(* CoDeSys 2.3.9.41 project: dct.pro *)
(* Libraries: STANDARD.LIB 4.10.05 11:14:46, IECSFC.LIB 13.4.06 15:51:28, SYSLIBTIME.LIB 20.2.06 13:31:16, SYSTASKINFO.LIB 20.2.06 13:31:38, ANALYZATION.LIB 5.10.99 09:05:06, SYSLIBCALLBACK.LIB 20.2.06 13:31:08 *)

(* PLC configuration (modules and I/O channels)
Discrete input 6 bit [ID100] node 0, in %IB0 out %QB0 {Filtrationtime = 10; Filtrationtime = 10; Filtrationtime = 10; Filtrationtime = 10; Filtrationtime = 10; Filtrationtime = 10; Visibility = No; PinCount = 6; WatchDogPeriod = 1000; PollPeriod = 1}
  AT %IX0.0 [BitInput]
  AT %IX0.1 [BitInput]
  AT %IX0.2 [BitInput]
  AT %IX0.3 [BitInput]
  AT %IX0.4 [BitInput]
  AT %IX0.5 [BitInput]
vuh1 AT %QX1.0 [BitOutput]
vuh2 AT %QX1.1 [BitOutput]
vuh31 AT %QX1.2 [BitOutput]
vuh4 AT %QX1.3 [BitOutput]
Special output [ID104] node 2, in %IB2 out %QB2 {Visibility = No; PinCount = 1}
  AT %QX2.0 [BitOutput] Special output
Unifed signal sensor [ID700] node 3, in %IB3 out %QB3 {Type_of_sensor700 = IT_0_20; measure_interval = 0.5; ainlow = 0; ainhigh = 20; first_cor_point = 0; first_delta = 0; second_cor_point = 0; second_delta = 0; third_cor_point = 0; third_delta = 0; Visibility = No}
  AT %ID3.0 [FloatInput] Value
  AT %IW3.1 [WordInput] Circular time
  Analog Input [ID107] node 0, in %IB3.0 out %QB3.0
Unifed signal sensor [ID700] node 4, in %IB4 out %QB4 {Type_of_sensor700 = IT_0_20; measure_interval = 0.5; ainlow = 0; ainhigh = 20; first_cor_point = 0; first_delta = 0; second_cor_point = 0; second_delta = 0; third_cor_point = 0; third_delta = 0; Visibility = No}
  AT %ID4.0 [FloatInput] Value
  AT %IW4.1 [WordInput] Circular time
  Analog Input [ID107] node 0, in %IB4.0 out %QB4.0
Unifed signal sensor [ID700] node 5, in %IB5 out %QB5 {Type_of_sensor700 = IT_0_20; measure_interval = 0.5; ainlow = 0; ainhigh = 20; first_cor_point = 0; first_delta = 0; second_cor_point = 0; second_delta = 0; third_cor_point = 0; third_delta = 0; Visibility = No}
  AT %ID5.0 [FloatInput] Value
  AT %IW5.1 [WordInput] Circular time
  Analog Input [ID107] node 0, in %IB5.0 out %QB5.0
Unifed signal sensor [ID700] node 6, in %IB6 out %QB6 {Type_of_sensor700 = IT_0_20; measure_interval = 0.5; ainlow = 0; ainhigh = 20; first_cor_point = 0; first_delta = 0; second_cor_point = 0; second_delta = 0; third_cor_point = 0; third_delta = 0; Visibility = No}
  AT %ID6.0 [FloatInput] Value
  AT %IW6.1 [WordInput] Circular time
  Analog Input [ID107] node 0, in %IB6.0 out %QB6.0
Analog output [ID106] node 7, in %IB7 out %QB7 {DAC_Type = Voltage 0-10 B; Analog_offset_correction = 0; Analog_full_range_correction = 0; SafeValueFloat = 0; Visibility = No}
  AT %QD7.0 [FloatOutput] Value
  AT %QD8.0 [FloatOutput] Value
AT %QD9.0 [DWordOutput] Last address
AT %QW9.1 [WordOutput] Last error
RS-485-1 [COM1_USART] node 0, in %IB9.0 out %QB9.0 {CommunicationSpeed = 11520; Parity = NO PARITY CHECK; BitLength = 8 bits; StopLength = One stop bit; InterfaceType = RS485; FrameOriented = RTU; Timeout = 0; Visibility = No}
AT %QB9.1.0 [ComChannel] Command (0xff - Start)
AT %IB9.1.0.0 [ByteInput]
MKV1 AT %QW9.1.1.0 [WordOutput]
MKV2 AT %QW9.1.2.0 [WordOutput]
MKV3 AT %QW9.1.3.0 [WordOutput]
MKV4 AT %QW9.1.4.0 [WordOutput]
TCP [TCP_ID221] node 0, in %IB10.0.0 out %QB10.0.0 {RemotePort = 502; Visibility = Yes}
AT %QB10.1.0 [ByteOutput]
AT %QB10.2.0 [ByteOutput]
*)

(* POU PLC_PRG, SFC *)
PROGRAM PLC_PRG
VAR
	pusk: BOOL;(*local PUSK CoDeSys*)
	bb: BOOL;(*zminna perehodu*)
	rs1: RS;(*reset set*)
	t1: TON;(*timer*)
	t22: TON;(*timer*)
	t11: TON;(*timer*)
	nn: BOOL;(*zminna zapusku kroku*)
	kl: BOOL;(*zminna zapusku kroku*)
	gh: BOOL;(*zminna zapusku kroku*)
	t: TON;(*timer*)
	t33: TON;(*timer*)
	t55: TON;(*timer*)
	tt45: TON;(*timer*)
	simp01: BOOL;(*zmina dlya SIMPLE SCADA*)
	simp11: BOOL;(*zmina dlya SIMPLE SCADA*)
	simp21: BOOL;(*zmina dlya SIMPLE SCADA*)
	simp31: BOOL;(*zmina dlya SIMPLE SCADA*)
	simp41: BOOL;(*zmina dlya SIMPLE SCADA*)
	simp61: BOOL;(*zmina dlya SIMPLE SCADA*)
	simp71: BOOL;(*zmina dlya SIMPLE SCADA*)
	simp81: BOOL;(*zmina dlya SIMPLE SCADA*)
	ttt: TON;(*timer*)
	tttt: TON;(*timer*)
	t123: TON;(*timer*)
	tt3: TON;(*timer*)
	dd: BOOL;(*zminna zapusku kroku*)
	tttttt: TON;(*timer*)
	t567: TON;(*timer*)
	pp: BOOL;(*zminna perehodu*)
	ts1: BOOL;(*zmina dlya TRACE MODE6*)
	ts8: BOOL;(*zmina dlya TRACE MODE6*)
	ts2: BOOL;(*zmina dlya TRACE MODE6*)
	ts3: BOOL;(*zmina dlya TRACE MODE6*)
	ts4: BOOL;(*zmina dlya TRACE MODE6*)
	tonnnn: TON;(*timer*)
	tank: BOOL;(*zminna perehodu*)
	tf1: TOF;(*timer*)
	tn2: TON;(*timer*)
	tyu: TON;(*timer*)
	jhg: BOOL;(*zminna zapusku kroku*)
END_VAR
VAR (* helpers for the ST form of the networks *)
	_t10 : BOOL;
	_en1 : BOOL;
	_t1 : BOOL;
	_t7 : BOOL;
	_t1_ : BOOL;
	_t12 : BOOL;
	_t2 : BOOL;
	_en1_ : BOOL;
	_t1__ : BOOL;
	_t1___ : BOOL;
	_en1__ : BOOL;
	_t1____ : BOOL;
END_VAR
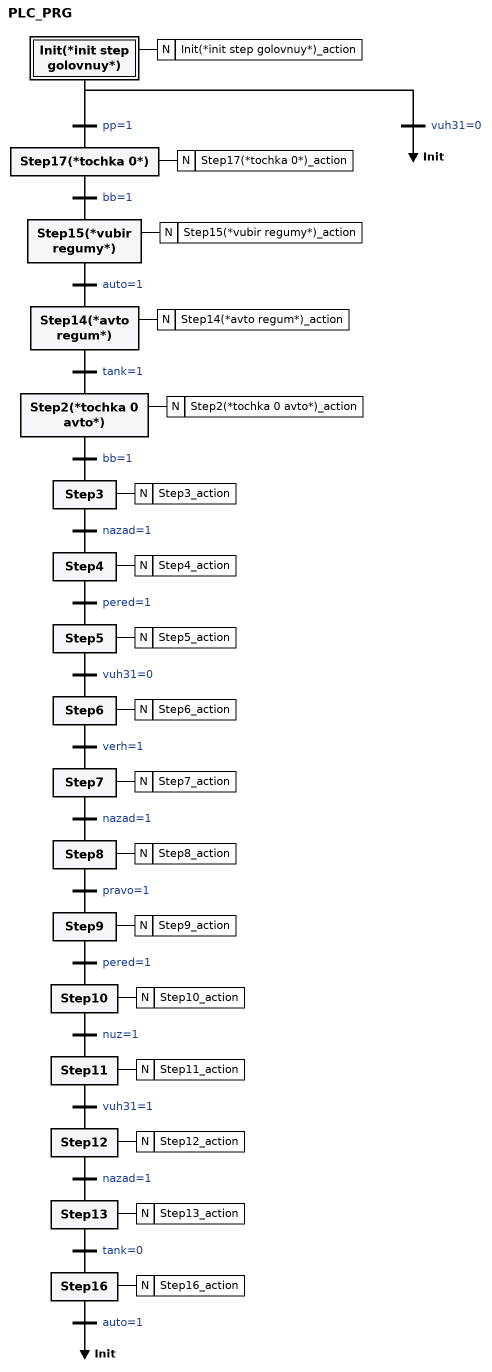
INITIAL_STEP Init(*init step golovnuy*):
	Init(*init step golovnuy*)_action(N);
END_STEP
TRANSITION FROM Init(*init step golovnuy*) TO Step17(*tochka 0*) := pp=1;
END_TRANSITION
TRANSITION FROM Init(*init step golovnuy*) TO Init := vuh31=0;
END_TRANSITION
STEP Step17(*tochka 0*):
	Step17(*tochka 0*)_action(N);
END_STEP
TRANSITION FROM Step17(*tochka 0*) TO Step15(*vubir regumy*) := bb=1;
END_TRANSITION
STEP Step15(*vubir regumy*):
	Step15(*vubir regumy*)_action(N);
END_STEP
TRANSITION FROM Step15(*vubir regumy*) TO Step14(*avto regum*) := auto=1;
END_TRANSITION
STEP Step14(*avto regum*):
	Step14(*avto regum*)_action(N);
END_STEP
TRANSITION FROM Step14(*avto regum*) TO Step2(*tochka 0 avto*) := tank=1;
END_TRANSITION
STEP Step2(*tochka 0 avto*):
	Step2(*tochka 0 avto*)_action(N);
END_STEP
TRANSITION FROM Step2(*tochka 0 avto*) TO Step3 := bb=1;
END_TRANSITION
STEP Step3:
	Step3_action(N);
END_STEP
TRANSITION FROM Step3 TO Step4 := nazad=1;
END_TRANSITION
STEP Step4:
	Step4_action(N);
END_STEP
TRANSITION FROM Step4 TO Step5 := pered=1;
END_TRANSITION
STEP Step5:
	Step5_action(N);
END_STEP
TRANSITION FROM Step5 TO Step6 := vuh31=0;
END_TRANSITION
STEP Step6:
	Step6_action(N);
END_STEP
TRANSITION FROM Step6 TO Step7 := verh=1;
END_TRANSITION
STEP Step7:
	Step7_action(N);
END_STEP
TRANSITION FROM Step7 TO Step8 := nazad=1;
END_TRANSITION
STEP Step8:
	Step8_action(N);
END_STEP
TRANSITION FROM Step8 TO Step9 := pravo=1;
END_TRANSITION
STEP Step9:
	Step9_action(N);
END_STEP
TRANSITION FROM Step9 TO Step10 := pered=1;
END_TRANSITION
STEP Step10:
	Step10_action(N);
END_STEP
TRANSITION FROM Step10 TO Step11 := nuz=1;
END_TRANSITION
STEP Step11:
	Step11_action(N);
END_STEP
TRANSITION FROM Step11 TO Step12 := vuh31=1;
END_TRANSITION
STEP Step12:
	Step12_action(N);
END_STEP
TRANSITION FROM Step12 TO Step13 := nazad=1;
END_TRANSITION
STEP Step13:
	Step13_action(N);
END_STEP
TRANSITION FROM Step13 TO Step16 := tank=0;
END_TRANSITION
STEP Step16:
	Step16_action(N);
END_STEP
TRANSITION FROM Step16 TO Init := auto=1;
END_TRANSITION

ACTION Init(*init step golovnuy*)_action:
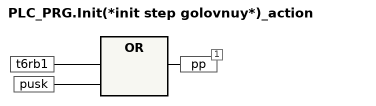
_CFC_ (* Continuous Function Chart, elements in execution order *)
#0 OR(t6rb1, pusk)
#1 pp <= #0
_END_CFC_
(* the same logic as Structured Text *)
pp := t6rb1 OR pusk;
END_ACTION

ACTION Step17(*tochka 0*)_action:
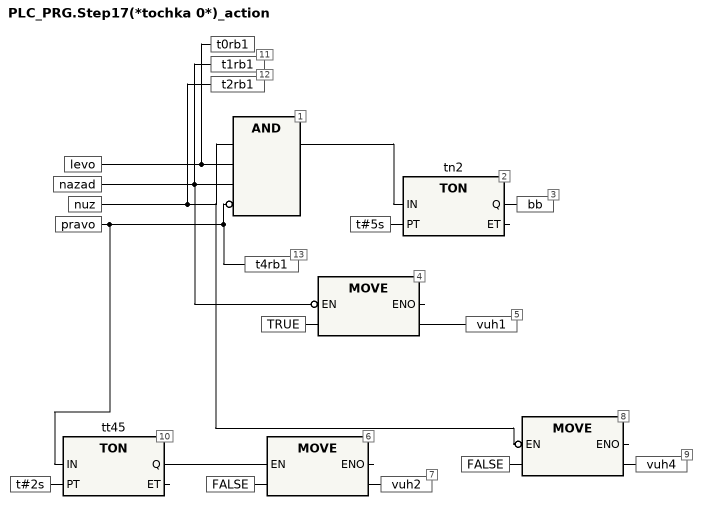
_CFC_ (* Continuous Function Chart, elements in execution order *)
#0 t0rb1 <= levo
#1 AND(nuz, levo, nazad, NOT pravo)
#2 tn2:TON(IN: #1, PT: t#5s)
#3 bb <= #2.Q
#4 MOVE(EN: NOT nazad, TRUE)
#5 vuh1 <= #4
#6 MOVE(EN: #10.Q, FALSE)
#7 vuh2 <= #6
#8 MOVE(EN: NOT nuz, FALSE)
#9 vuh4 <= #8
#10 tt45:TON(IN: pravo, PT: t#2s)
#11 t1rb1 <= nazad
#12 t2rb1 <= nuz
#13 t4rb1 <= pravo
_END_CFC_
(* the same logic as Structured Text *)
t0rb1 := levo;
tn2(IN := nuz AND levo AND nazad AND NOT pravo, PT := t#5s);
bb := tn2.Q;
IF NOT nazad THEN vuh1 := TRUE; END_IF;
IF tt45.Q THEN vuh2 := FALSE; END_IF;
IF NOT nuz THEN vuh4 := FALSE; END_IF;
tt45(IN := pravo, PT := t#2s);
t1rb1 := nazad;
t2rb1 := nuz;
t4rb1 := pravo;
END_ACTION

ACTION Step15(*vubir regumy*)_action:
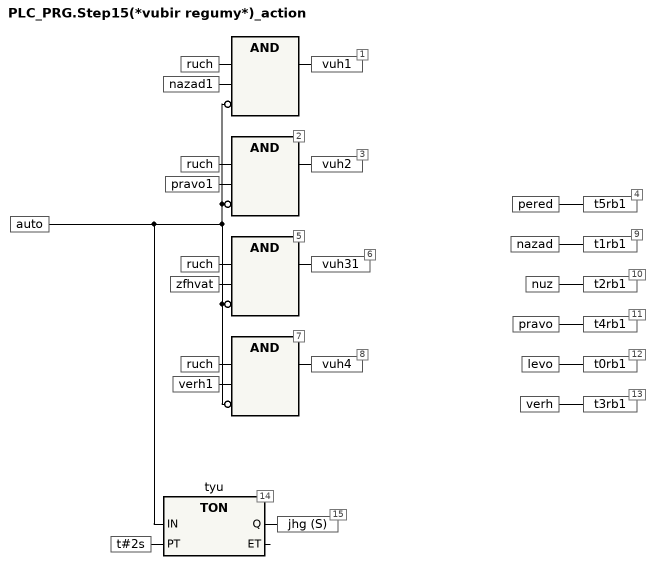
_CFC_ (* Continuous Function Chart, elements in execution order *)
#0 AND(ruch, nazad1, NOT auto)
#1 vuh1 <= #0
#2 AND(ruch, pravo1, NOT auto)
#3 vuh2 <= #2
#4 t5rb1 <= pered
#5 AND(ruch, zfhvat, NOT auto)
#6 vuh31 <= #5
#7 AND(ruch, verh1, NOT auto)
#8 vuh4 <= #7
#9 t1rb1 <= nazad
#10 t2rb1 <= nuz
#11 t4rb1 <= pravo
#12 t0rb1 <= levo
#13 t3rb1 <= verh
#14 tyu:TON(IN: auto, PT: t#2s)
#15 S jhg <= #14.Q
_END_CFC_
(* the same logic as Structured Text *)
vuh1 := ruch AND nazad1 AND NOT auto;
vuh2 := ruch AND pravo1 AND NOT auto;
t5rb1 := pered;
vuh31 := ruch AND zfhvat AND NOT auto;
vuh4 := ruch AND verh1 AND NOT auto;
t1rb1 := nazad;
t2rb1 := nuz;
t4rb1 := pravo;
t0rb1 := levo;
t3rb1 := verh;
tyu(IN := auto, PT := t#2s);
IF tyu.Q THEN jhg := TRUE; END_IF;
END_ACTION

ACTION Step14(*avto regum*)_action:
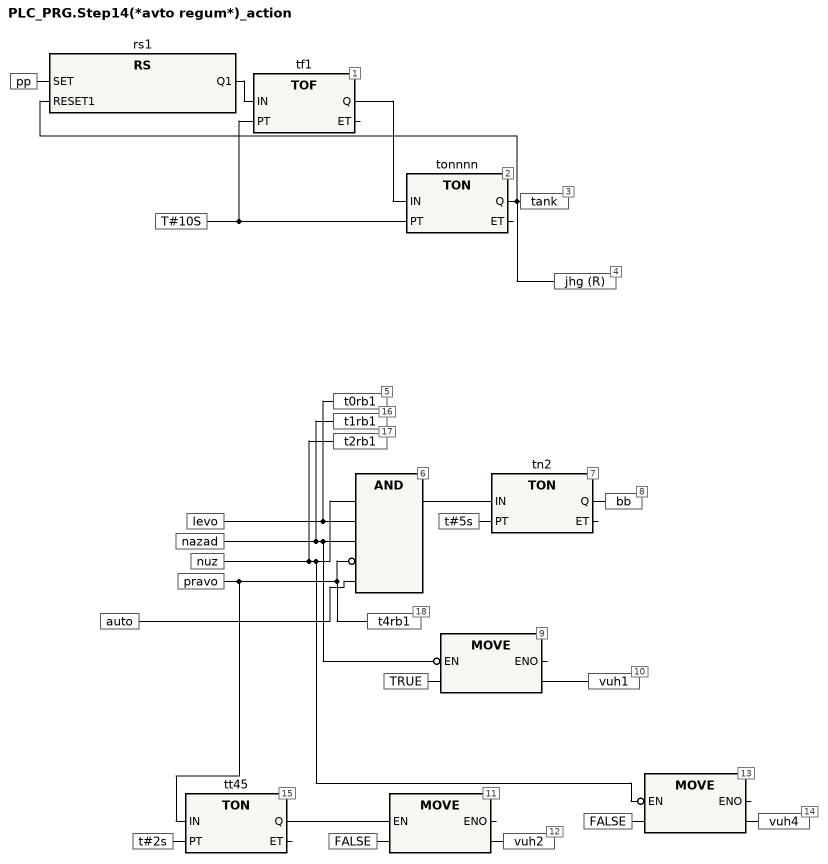
_CFC_ (* Continuous Function Chart, elements in execution order *)
#0 rs1:RS(SET: pp, RESET1: #2.Q)
#1 tf1:TOF(IN: #0.Q1, PT: T#10S)
#2 tonnnn:TON(IN: #1.Q, PT: T#10S)
#3 tank <= #2.Q
#4 R jhg <= #2.Q
#5 t0rb1 <= levo
#6 AND(nuz, levo, nazad, NOT pravo, auto)
#7 tn2:TON(IN: #6, PT: t#5s)
#8 bb <= #7.Q
#9 MOVE(EN: NOT nazad, TRUE)
#10 vuh1 <= #9
#11 MOVE(EN: #15.Q, FALSE)
#12 vuh2 <= #11
#13 MOVE(EN: NOT nuz, FALSE)
#14 vuh4 <= #13
#15 tt45:TON(IN: pravo, PT: t#2s)
#16 t1rb1 <= nazad
#17 t2rb1 <= nuz
#18 t4rb1 <= pravo
_END_CFC_
(* the same logic as Structured Text *)
rs1(SET := pp, RESET1 := tonnnn.Q);
tf1(IN := rs1.Q1, PT := T#10S);
tonnnn(IN := tf1.Q, PT := T#10S);
tank := tonnnn.Q;
IF tonnnn.Q THEN jhg := FALSE; END_IF;
t0rb1 := levo;
tn2(IN := nuz AND levo AND nazad AND NOT pravo AND auto, PT := t#5s);
bb := tn2.Q;
IF NOT nazad THEN vuh1 := TRUE; END_IF;
IF tt45.Q THEN vuh2 := FALSE; END_IF;
IF NOT nuz THEN vuh4 := FALSE; END_IF;
tt45(IN := pravo, PT := t#2s);
t1rb1 := nazad;
t2rb1 := nuz;
t4rb1 := pravo;
END_ACTION

ACTION Step2(*tochka 0 avto*)_action:
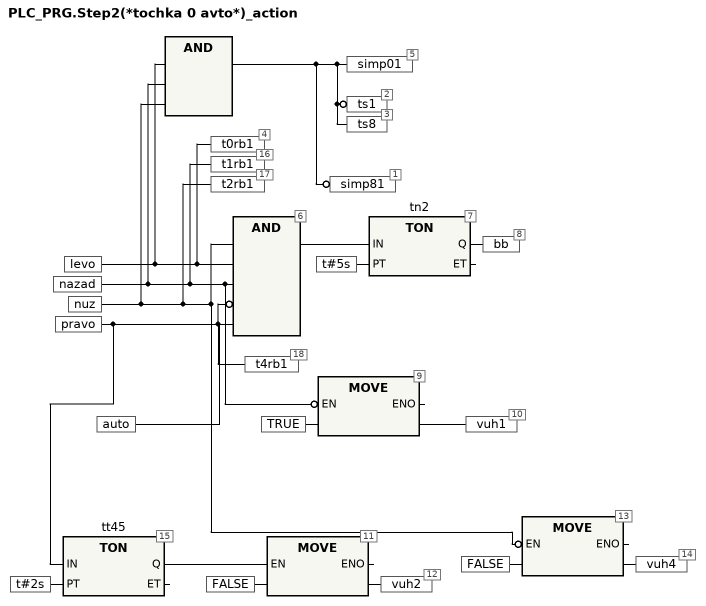
_CFC_ (* Continuous Function Chart, elements in execution order *)
#0 AND(levo, nazad, nuz)
#1 simp81 <= NOT #0
#2 ts1 <= NOT #0
#3 ts8 <= #0
#4 t0rb1 <= levo
#5 simp01 <= #0
#6 AND(nuz, levo, nazad, NOT pravo, auto)
#7 tn2:TON(IN: #6, PT: t#5s)
#8 bb <= #7.Q
#9 MOVE(EN: NOT nazad, TRUE)
#10 vuh1 <= #9
#11 MOVE(EN: #15.Q, FALSE)
#12 vuh2 <= #11
#13 MOVE(EN: NOT nuz, FALSE)
#14 vuh4 <= #13
#15 tt45:TON(IN: pravo, PT: t#2s)
#16 t1rb1 <= nazad
#17 t2rb1 <= nuz
#18 t4rb1 <= pravo
_END_CFC_
(* the same logic as Structured Text *)
simp81 := NOT (levo AND nazad AND nuz);
ts1 := NOT (levo AND nazad AND nuz);
ts8 := levo AND nazad AND nuz;
t0rb1 := levo;
simp01 := levo AND nazad AND nuz;
tn2(IN := nuz AND levo AND nazad AND NOT pravo AND auto, PT := t#5s);
bb := tn2.Q;
IF NOT nazad THEN vuh1 := TRUE; END_IF;
IF tt45.Q THEN vuh2 := FALSE; END_IF;
IF NOT nuz THEN vuh4 := FALSE; END_IF;
tt45(IN := pravo, PT := t#2s);
t1rb1 := nazad;
t2rb1 := nuz;
t4rb1 := pravo;
END_ACTION

ACTION Step3_action:
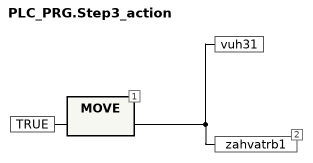
_CFC_ (* Continuous Function Chart, elements in execution order *)
#0 vuh31 <= #1
#1 MOVE(TRUE)
#2 zahvatrb1 <= #1
_END_CFC_
(* the same logic as Structured Text *)
vuh31 := _t10;
_t10 := TRUE;
zahvatrb1 := _t10;
END_ACTION

ACTION Step4_action:
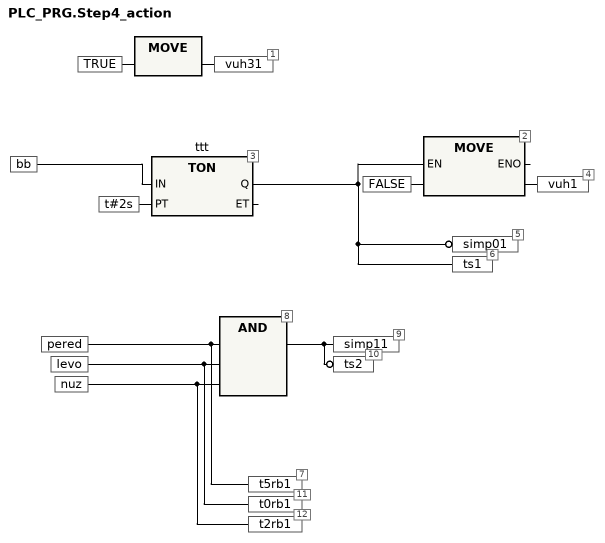
_CFC_ (* Continuous Function Chart, elements in execution order *)
#0 MOVE(TRUE)
#1 vuh31 <= #0
#2 MOVE(EN: #3.Q, FALSE)
#3 ttt:TON(IN: bb, PT: t#2s)
#4 vuh1 <= #2
#5 simp01 <= NOT #3.Q
#6 ts1 <= #3.Q
#7 t5rb1 <= pered
#8 AND(pered, levo, nuz)
#9 simp11 <= #8
#10 ts2 <= NOT #8
#11 t0rb1 <= levo
#12 t2rb1 <= nuz
_END_CFC_
(* the same logic as Structured Text *)
vuh31 := TRUE;
_en1 := ttt.Q;
IF _en1 THEN _t1 := FALSE; END_IF;
ttt(IN := bb, PT := t#2s);
IF _en1 THEN vuh1 := _t1; END_IF;
simp01 := NOT ttt.Q;
ts1 := ttt.Q;
t5rb1 := pered;
simp11 := pered AND levo AND nuz;
ts2 := NOT (pered AND levo AND nuz);
t0rb1 := levo;
t2rb1 := nuz;
END_ACTION

ACTION Step5_action:
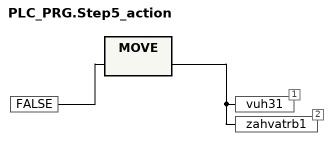
_CFC_ (* Continuous Function Chart, elements in execution order *)
#0 MOVE(FALSE)
#1 vuh31 <= #0
#2 zahvatrb1 <= #0
_END_CFC_
(* the same logic as Structured Text *)
vuh31 := FALSE;
zahvatrb1 := FALSE;
END_ACTION

ACTION Step6_action:
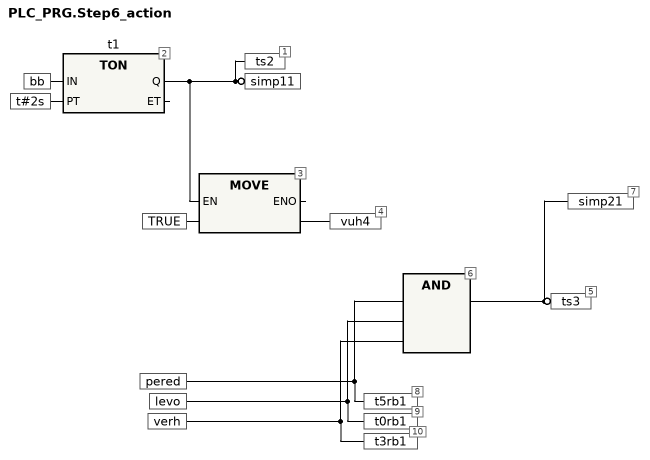
_CFC_ (* Continuous Function Chart, elements in execution order *)
#0 simp11 <= NOT #2.Q
#1 ts2 <= #2.Q
#2 t1:TON(IN: bb, PT: t#2s)
#3 MOVE(EN: #2.Q, TRUE)
#4 vuh4 <= #3
#5 ts3 <= NOT #6
#6 AND(pered, levo, verh)
#7 simp21 <= #6
#8 t5rb1 <= pered
#9 t0rb1 <= levo
#10 t3rb1 <= verh
_END_CFC_
(* the same logic as Structured Text *)
simp11 := NOT t1.Q;
ts2 := t1.Q;
t1(IN := bb, PT := t#2s);
IF t1.Q THEN vuh4 := TRUE; END_IF;
ts3 := NOT _t7;
_t7 := pered AND levo AND verh;
simp21 := _t7;
t5rb1 := pered;
t0rb1 := levo;
t3rb1 := verh;
END_ACTION

ACTION Step7_action:
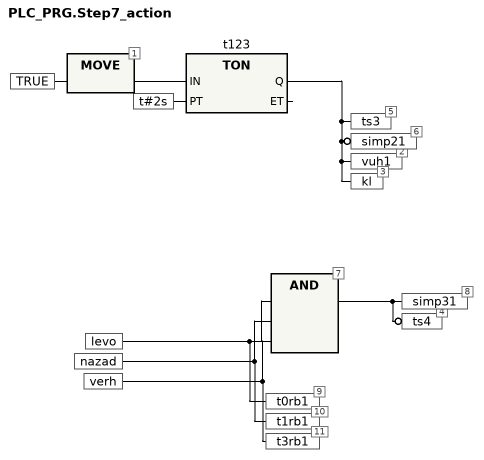
_CFC_ (* Continuous Function Chart, elements in execution order *)
#0 t123:TON(IN: #1, PT: t#2s)
#1 MOVE(TRUE)
#2 vuh1 <= #0.Q
#3 kl <= #0.Q
#4 ts4 <= NOT #7
#5 ts3 <= #0.Q
#6 simp21 <= NOT #0.Q
#7 AND(levo, nazad, verh)
#8 simp31 <= #7
#9 t0rb1 <= levo
#10 t1rb1 <= nazad
#11 t3rb1 <= verh
_END_CFC_
(* the same logic as Structured Text *)
t123(IN := _t1_, PT := t#2s);
_t1_ := TRUE;
vuh1 := t123.Q;
kl := t123.Q;
ts4 := NOT _t12;
ts3 := t123.Q;
simp21 := NOT t123.Q;
_t12 := levo AND nazad AND verh;
simp31 := _t12;
t0rb1 := levo;
t1rb1 := nazad;
t3rb1 := verh;
END_ACTION

ACTION Step8_action:
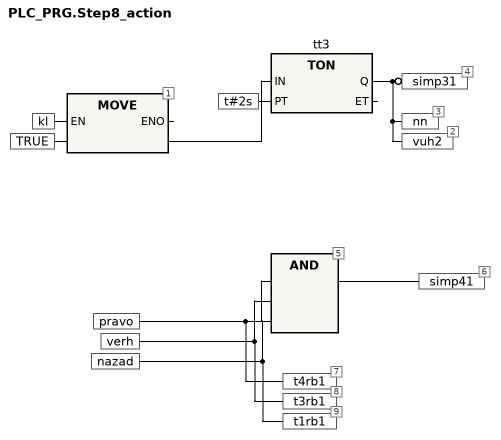
_CFC_ (* Continuous Function Chart, elements in execution order *)
#0 tt3:TON(IN: #1, PT: t#2s)
#1 MOVE(EN: kl, TRUE)
#2 vuh2 <= #0.Q
#3 nn <= #0.Q
#4 simp31 <= NOT #0.Q
#5 AND(pravo, verh, nazad)
#6 simp41 <= #5
#7 t4rb1 <= pravo
#8 t3rb1 <= verh
#9 t1rb1 <= nazad
_END_CFC_
(* the same logic as Structured Text *)
tt3(IN := _t2, PT := t#2s);
IF kl THEN _t2 := TRUE; END_IF;
vuh2 := tt3.Q;
nn := tt3.Q;
simp31 := NOT tt3.Q;
simp41 := pravo AND verh AND nazad;
t4rb1 := pravo;
t3rb1 := verh;
t1rb1 := nazad;
END_ACTION

ACTION Step9_action:
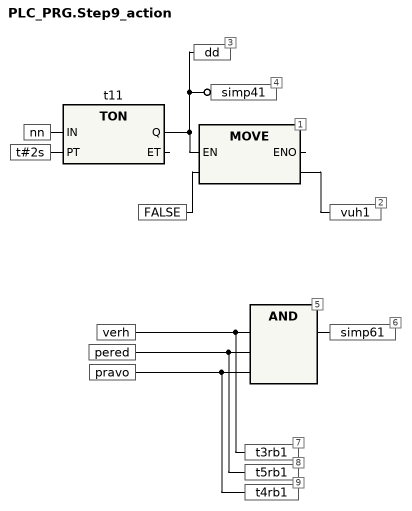
_CFC_ (* Continuous Function Chart, elements in execution order *)
#0 t11:TON(IN: nn, PT: t#2s)
#1 MOVE(EN: #0.Q, FALSE)
#2 vuh1 <= #1
#3 dd <= #0.Q
#4 simp41 <= NOT #0.Q
#5 AND(verh, pered, pravo)
#6 simp61 <= #5
#7 t3rb1 <= verh
#8 t5rb1 <= pered
#9 t4rb1 <= pravo
_END_CFC_
(* the same logic as Structured Text *)
t11(IN := nn, PT := t#2s);
IF t11.Q THEN vuh1 := FALSE; END_IF;
dd := t11.Q;
simp41 := NOT t11.Q;
simp61 := verh AND pered AND pravo;
t3rb1 := verh;
t5rb1 := pered;
t4rb1 := pravo;
END_ACTION

ACTION Step10_action:
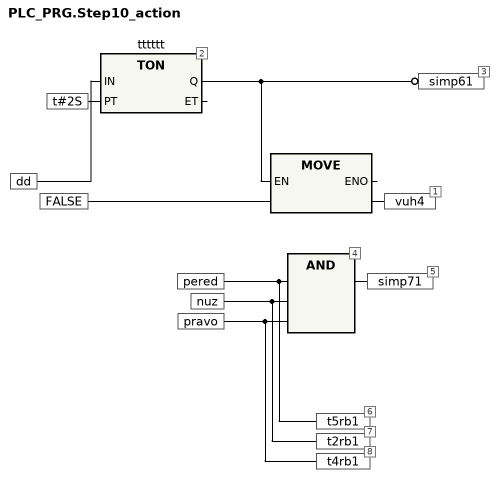
_CFC_ (* Continuous Function Chart, elements in execution order *)
#0 MOVE(EN: #2.Q, FALSE)
#1 vuh4 <= #0
#2 tttttt:TON(IN: dd, PT: t#2S)
#3 simp61 <= NOT #2.Q
#4 AND(pered, nuz, pravo)
#5 simp71 <= #4
#6 t5rb1 <= pered
#7 t2rb1 <= nuz
#8 t4rb1 <= pravo
_END_CFC_
(* the same logic as Structured Text *)
IF tttttt.Q THEN vuh4 := FALSE; END_IF;
tttttt(IN := dd, PT := t#2S);
simp61 := NOT tttttt.Q;
simp71 := pered AND nuz AND pravo;
t5rb1 := pered;
t2rb1 := nuz;
t4rb1 := pravo;
END_ACTION

ACTION Step11_action:
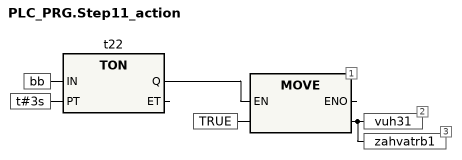
_CFC_ (* Continuous Function Chart, elements in execution order *)
#0 t22:TON(IN: bb, PT: t#3s)
#1 MOVE(EN: #0.Q, TRUE)
#2 vuh31 <= #1
#3 zahvatrb1 <= #1
_END_CFC_
(* the same logic as Structured Text *)
t22(IN := bb, PT := t#3s);
_en1_ := t22.Q;
IF _en1_ THEN _t1__ := TRUE; END_IF;
IF _en1_ THEN vuh31 := _t1__; END_IF;
IF _en1_ THEN zahvatrb1 := _t1__; END_IF;
END_ACTION

ACTION Step12_action:
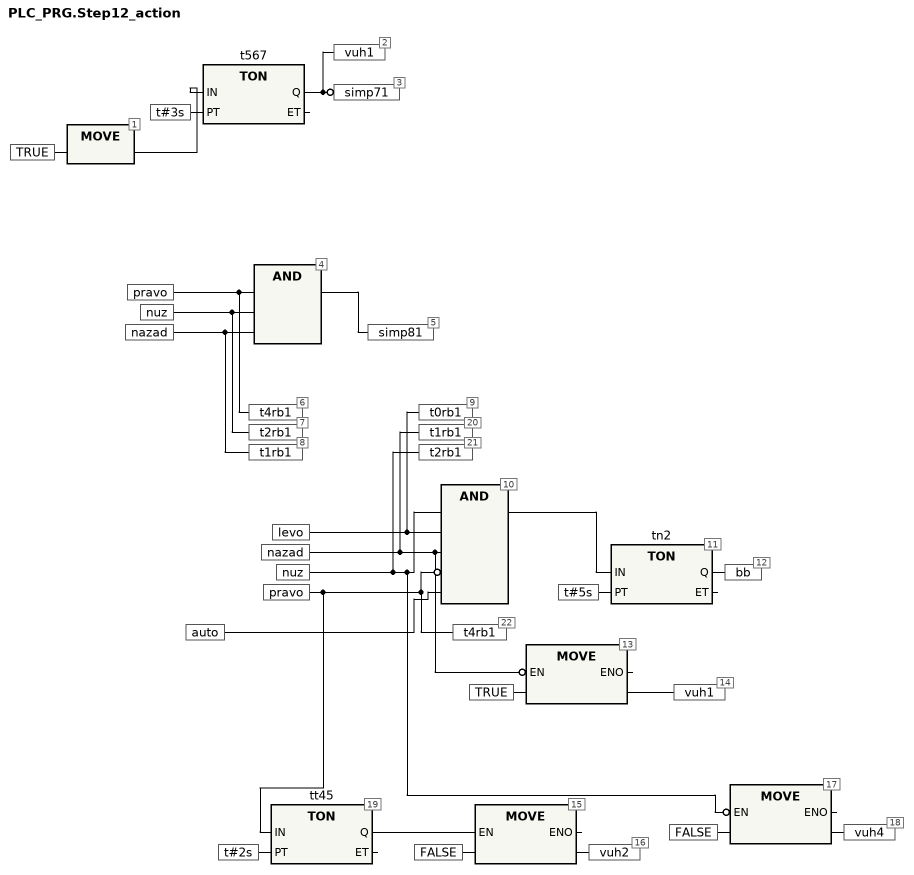
_CFC_ (* Continuous Function Chart, elements in execution order *)
#0 t567:TON(IN: #1, PT: t#3s)
#1 MOVE(TRUE)
#2 vuh1 <= #0.Q
#3 simp71 <= NOT #0.Q
#4 AND(pravo, nuz, nazad)
#5 simp81 <= #4
#6 t4rb1 <= pravo
#7 t2rb1 <= nuz
#8 t1rb1 <= nazad
#9 t0rb1 <= levo
#10 AND(nuz, levo, nazad, NOT pravo, auto)
#11 tn2:TON(IN: #10, PT: t#5s)
#12 bb <= #11.Q
#13 MOVE(EN: NOT nazad, TRUE)
#14 vuh1 <= #13
#15 MOVE(EN: #19.Q, FALSE)
#16 vuh2 <= #15
#17 MOVE(EN: NOT nuz, FALSE)
#18 vuh4 <= #17
#19 tt45:TON(IN: pravo, PT: t#2s)
#20 t1rb1 <= nazad
#21 t2rb1 <= nuz
#22 t4rb1 <= pravo
_END_CFC_
(* the same logic as Structured Text *)
t567(IN := _t1___, PT := t#3s);
_t1___ := TRUE;
vuh1 := t567.Q;
simp71 := NOT t567.Q;
simp81 := pravo AND nuz AND nazad;
t4rb1 := pravo;
t2rb1 := nuz;
t1rb1 := nazad;
t0rb1 := levo;
tn2(IN := nuz AND levo AND nazad AND NOT pravo AND auto, PT := t#5s);
bb := tn2.Q;
IF NOT nazad THEN vuh1 := TRUE; END_IF;
IF tt45.Q THEN vuh2 := FALSE; END_IF;
IF NOT nuz THEN vuh4 := FALSE; END_IF;
tt45(IN := pravo, PT := t#2s);
t1rb1 := nazad;
t2rb1 := nuz;
t4rb1 := pravo;
END_ACTION

ACTION Step13_action:
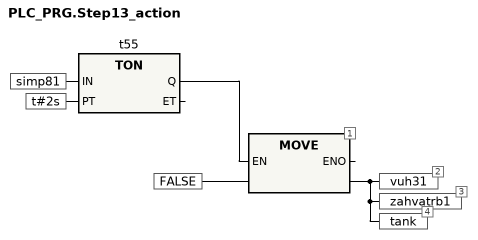
_CFC_ (* Continuous Function Chart, elements in execution order *)
#0 t55:TON(IN: simp81, PT: t#2s)
#1 MOVE(EN: #0.Q, FALSE)
#2 vuh31 <= #1
#3 zahvatrb1 <= #1
#4 tank <= #1
_END_CFC_
(* the same logic as Structured Text *)
t55(IN := simp81, PT := t#2s);
_en1__ := t55.Q;
IF _en1__ THEN _t1____ := FALSE; END_IF;
IF _en1__ THEN vuh31 := _t1____; END_IF;
IF _en1__ THEN zahvatrb1 := _t1____; END_IF;
IF _en1__ THEN tank := _t1____; END_IF;
END_ACTION

ACTION Step16_action:
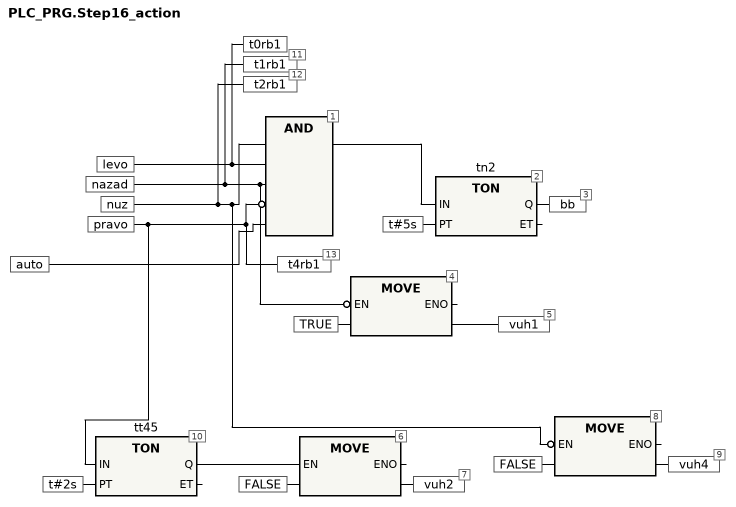
_CFC_ (* Continuous Function Chart, elements in execution order *)
#0 t0rb1 <= levo
#1 AND(nuz, levo, nazad, NOT pravo, auto)
#2 tn2:TON(IN: #1, PT: t#5s)
#3 bb <= #2.Q
#4 MOVE(EN: NOT nazad, TRUE)
#5 vuh1 <= #4
#6 MOVE(EN: #10.Q, FALSE)
#7 vuh2 <= #6
#8 MOVE(EN: NOT nuz, FALSE)
#9 vuh4 <= #8
#10 tt45:TON(IN: pravo, PT: t#2s)
#11 t1rb1 <= nazad
#12 t2rb1 <= nuz
#13 t4rb1 <= pravo
_END_CFC_
(* the same logic as Structured Text *)
t0rb1 := levo;
tn2(IN := nuz AND levo AND nazad AND NOT pravo AND auto, PT := t#5s);
bb := tn2.Q;
IF NOT nazad THEN vuh1 := TRUE; END_IF;
IF tt45.Q THEN vuh2 := FALSE; END_IF;
IF NOT nuz THEN vuh4 := FALSE; END_IF;
tt45(IN := pravo, PT := t#2s);
t1rb1 := nazad;
t2rb1 := nuz;
t4rb1 := pravo;
END_ACTION
END_PROGRAM

(* Visualisation fgdjgh
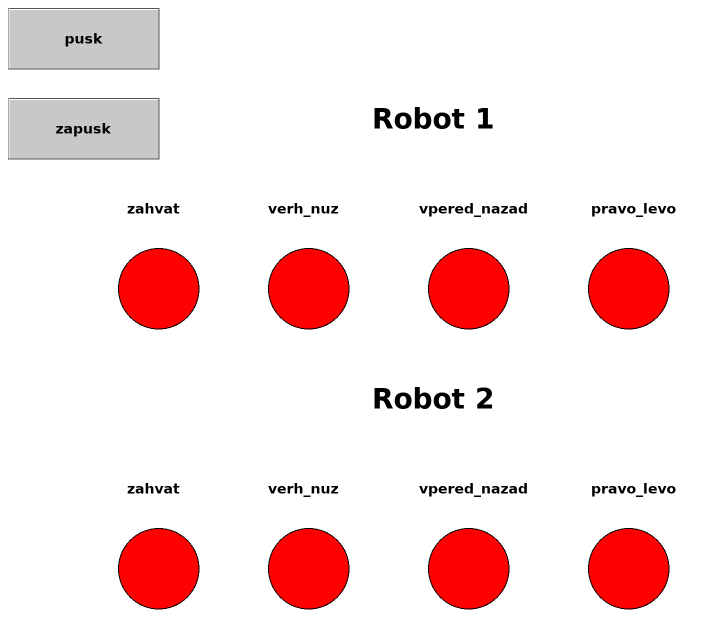
button at (70,20)-(221,81): text "pusk"; toggles PLC_PRG.pusk
button at (70,110)-(221,171): text "zapusk"; toggles PLC_PRG.zapusk
ellipse at (180,260)-(261,341): alarm colour if .vuh3
ellipse at (330,260)-(411,341): alarm colour if .vuh4
ellipse at (490,260)-(571,341): alarm colour if .vuh1
ellipse at (650,260)-(731,341): alarm colour if .vuh2
rectangle at (150,190)-(281,251): text "zahvat"
rectangle at (300,190)-(431,251): text "verh_nuz"
rectangle at (470,190)-(601,251): text "vpered_nazad"
rectangle at (630,190)-(761,251): text "pravo_levo"
rectangle at (280,90)-(711,171): text "Robot 1"
ellipse at (180,540)-(261,621): alarm colour if .MKV3
ellipse at (330,540)-(411,621): alarm colour if .MKV4
ellipse at (490,540)-(571,621): alarm colour if .MKV1
ellipse at (650,540)-(731,621): alarm colour if .MKV2
rectangle at (150,470)-(281,531): text "zahvat"
rectangle at (300,470)-(431,531): text "verh_nuz"
rectangle at (470,470)-(601,531): text "vpered_nazad"
rectangle at (630,470)-(761,531): text "pravo_levo"
rectangle at (280,370)-(711,451): text "Robot 2"
*)
